FUNCTION_BLOCK FB_System_BSp_Ablaufsteuerung
VAR_IN_OUT
	Zustand					: ST_System_BSp_Zustand;
	Stellwert				: ST_System_BSp_Stellwert;
	Steuerung				: ST_System_BSp_Steuerung;
END_VAR
VAR_INPUT
	Zustand_Stellventil		: ST_SV_Zustand;
	Zustand_Pumpe			: ST_PU_Zustand;
	Zustand_Pumpe_Sp		: ST_PU_Schuetz_Zustand;
END_VAR
VAR_OUTPUT
END_VAR
VAR
END_VAR

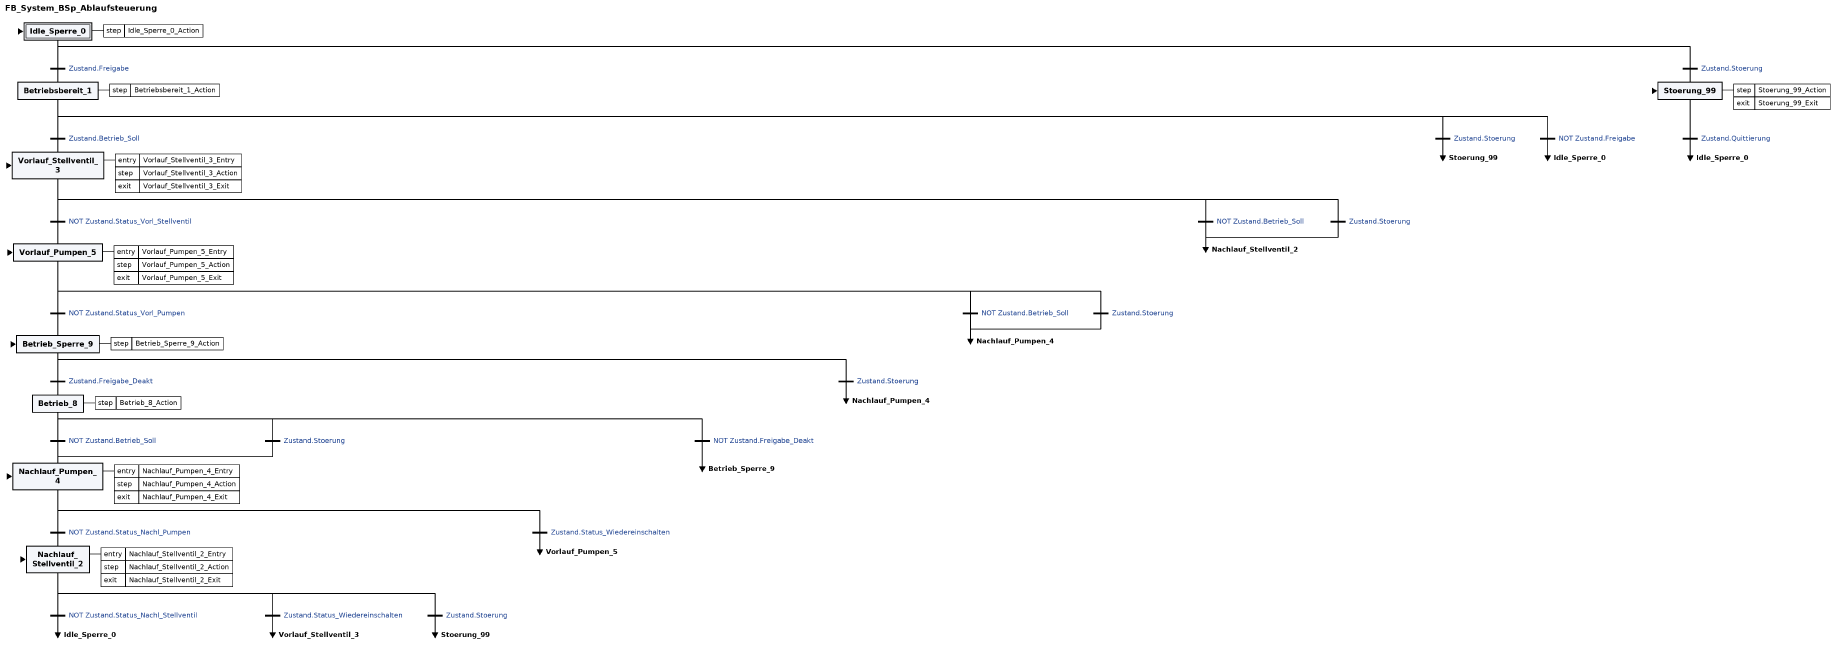
INITIAL_STEP Idle_Sperre_0:
    Idle_Sperre_0_Action(N);  // step action
END_STEP
TRANSITION FROM Idle_Sperre_0 TO Betriebsbereit_1
    := Zustand.Freigabe;
END_TRANSITION
TRANSITION FROM Idle_Sperre_0 TO Stoerung_99
    := Zustand.Stoerung;
END_TRANSITION
STEP Stoerung_99:
    Stoerung_99_Action(N);  // step action
    Stoerung_99_Exit(P0);  // exit action
END_STEP
TRANSITION FROM Stoerung_99 TO Idle_Sperre_0
    := Zustand.Quittierung;
END_TRANSITION
STEP Betriebsbereit_1:
    Betriebsbereit_1_Action(N);  // step action
END_STEP
TRANSITION FROM Betriebsbereit_1 TO Vorlauf_Stellventil_3
    := Zustand.Betrieb_Soll;
END_TRANSITION
TRANSITION FROM Betriebsbereit_1 TO Stoerung_99
    := Zustand.Stoerung;
END_TRANSITION
TRANSITION FROM Betriebsbereit_1 TO Idle_Sperre_0
    := NOT Zustand.Freigabe;
END_TRANSITION
STEP Vorlauf_Stellventil_3:
    Vorlauf_Stellventil_3_Entry(P1);  // entry action
    Vorlauf_Stellventil_3_Action(N);  // step action
    Vorlauf_Stellventil_3_Exit(P0);  // exit action
END_STEP
TRANSITION FROM Vorlauf_Stellventil_3 TO Vorlauf_Pumpen_5
    := NOT Zustand.Status_Vorl_Stellventil;
END_TRANSITION
TRANSITION FROM Vorlauf_Stellventil_3 TO Nachlauf_Stellventil_2
    := NOT Zustand.Betrieb_Soll;
END_TRANSITION
TRANSITION FROM Vorlauf_Stellventil_3 TO Nachlauf_Stellventil_2
    := Zustand.Stoerung;
END_TRANSITION
STEP Vorlauf_Pumpen_5:
    Vorlauf_Pumpen_5_Entry(P1);  // entry action
    Vorlauf_Pumpen_5_Action(N);  // step action
    Vorlauf_Pumpen_5_Exit(P0);  // exit action
END_STEP
TRANSITION FROM Vorlauf_Pumpen_5 TO Betrieb_Sperre_9
    := NOT Zustand.Status_Vorl_Pumpen;
END_TRANSITION
TRANSITION FROM Vorlauf_Pumpen_5 TO Nachlauf_Pumpen_4
    := NOT Zustand.Betrieb_Soll;
END_TRANSITION
TRANSITION FROM Vorlauf_Pumpen_5 TO Nachlauf_Pumpen_4
    := Zustand.Stoerung;
END_TRANSITION
STEP Betrieb_Sperre_9:
    Betrieb_Sperre_9_Action(N);  // step action
END_STEP
TRANSITION FROM Betrieb_Sperre_9 TO Betrieb_8
    := Zustand.Freigabe_Deakt;
END_TRANSITION
TRANSITION FROM Betrieb_Sperre_9 TO Nachlauf_Pumpen_4
    := Zustand.Stoerung;
END_TRANSITION
STEP Betrieb_8:
    Betrieb_8_Action(N);  // step action
END_STEP
TRANSITION FROM Betrieb_8 TO Nachlauf_Pumpen_4
    := NOT Zustand.Betrieb_Soll;
END_TRANSITION
TRANSITION FROM Betrieb_8 TO Nachlauf_Pumpen_4
    := Zustand.Stoerung;
END_TRANSITION
TRANSITION FROM Betrieb_8 TO Betrieb_Sperre_9
    := NOT Zustand.Freigabe_Deakt;
END_TRANSITION
STEP Nachlauf_Pumpen_4:
    Nachlauf_Pumpen_4_Entry(P1);  // entry action
    Nachlauf_Pumpen_4_Action(N);  // step action
    Nachlauf_Pumpen_4_Exit(P0);  // exit action
END_STEP
TRANSITION FROM Nachlauf_Pumpen_4 TO Nachlauf_Stellventil_2
    := NOT Zustand.Status_Nachl_Pumpen;
END_TRANSITION
TRANSITION FROM Nachlauf_Pumpen_4 TO Vorlauf_Pumpen_5
    := Zustand.Status_Wiedereinschalten;
END_TRANSITION
STEP Nachlauf_Stellventil_2:
    Nachlauf_Stellventil_2_Entry(P1);  // entry action
    Nachlauf_Stellventil_2_Action(N);  // step action
    Nachlauf_Stellventil_2_Exit(P0);  // exit action
END_STEP
TRANSITION FROM Nachlauf_Stellventil_2 TO Idle_Sperre_0
    := NOT Zustand.Status_Nachl_Stellventil;
END_TRANSITION
TRANSITION FROM Nachlauf_Stellventil_2 TO Vorlauf_Stellventil_3
    := Zustand.Status_Wiedereinschalten;
END_TRANSITION
TRANSITION FROM Nachlauf_Stellventil_2 TO Stoerung_99
    := Zustand.Stoerung;
END_TRANSITION

ACTION Betrieb_8_Action:
(* Stellwert setzen *)
Stellwert.Anford_Stellventil	:= TRUE;
Stellwert.Anford_Pumpe			:= TRUE;
Stellwert.Anford_Pumpe_Sp		:= TRUE;

(* Zustand setzen *)
Zustand.Status					:= E_System_BSp_Zustand_Status_Betrieb;
END_ACTION

ACTION Betrieb_Sperre_9_Action:
(* Stellwert setzen *)
Stellwert.Anford_Stellventil		:= TRUE;
Stellwert.Anford_Pumpe		:= TRUE;
Stellwert.Anford_Pumpe_Sp		:= TRUE;

(* Zustand setzen *)
Zustand.Status				:= E_System_BSp_Zustand_Status_Betrieb_Sperre;
END_ACTION

ACTION Betriebsbereit_1_Action:
(* Stellwert setzen *)
Stellwert.Anford_Stellventil	:= FALSE;
Stellwert.Anford_Pumpe			:= FALSE;
Stellwert.Anford_Pumpe_Sp		:= FALSE;

(* Zustand setzen *)
Zustand.Status			:= E_System_BSp_Zustand_Status_Betriebsbereit;
END_ACTION

ACTION Idle_Sperre_0_Action:
(* Stellwert setzen *)
Stellwert.Anford_Stellventil		:= FALSE;
Stellwert.Anford_Pumpe		:= FALSE;
Stellwert.Anford_Pumpe_Sp		:= FALSE;

(* Zustand setzen *)
Zustand.Status				:= E_System_BSp_Zustand_Status_Idle_Sperre;

(* Quittierungszustand auf False setzen, damit das System bei einer erneuten Störung nicht direkt wieder angeschaltet wird *)
Steuerung.Quittierung	:= FALSE;
END_ACTION

ACTION Nachlauf_Pumpen_4_Action:
(* Stellwert setzen *)
Stellwert.Anford_Stellventil	:= FALSE;
Stellwert.Anford_Pumpe			:= FALSE;
Stellwert.Anford_Pumpe_Sp		:= FALSE;

(* Zustand setzen *)
Zustand.Status				:= E_System_BSp_Zustand_Status_Nachl_Pumpen;
Zustand.Status_Nachl_Pumpen	:= Zustand_Pumpe.Betrieb OR Zustand_Pumpe_Sp.Betrieb OR Zustand_Pumpe.Status_Nachl OR Zustand_Pumpe_Sp.Status_Nachl;
Zustand.Status_Wiedereinschalten := Zustand.Betrieb_Soll AND Stellwert.Einschalten;
END_ACTION

ACTION Nachlauf_Pumpen_4_Entry:
Zustand.Status_Nachl_Pumpen	:= TRUE;
END_ACTION

ACTION Nachlauf_Pumpen_4_Exit:
Zustand.Status_Nachl_Pumpen	:= FALSE;
END_ACTION

ACTION Nachlauf_Stellventil_2_Action:
(* Stellwert setzen *)
Stellwert.Anford_Stellventil		:= FALSE;
Stellwert.Anford_Pumpe		:= FALSE;
Stellwert.Anford_Pumpe_Sp		:= FALSE;

(* Zustand setzen *)
Zustand.Status				:= E_System_BSp_Zustand_Status_Nachl_Stellventil;
Zustand.Status_Nachl_Stellventil	:= Zustand_Stellventil.Stellung OR Zustand_Stellventil.Stellungwechsel10;
Zustand.Status_Wiedereinschalten := Zustand.Betrieb_Soll AND Stellwert.Einschalten;
END_ACTION

ACTION Nachlauf_Stellventil_2_Entry:
Zustand.Status_Nachl_Stellventil	:= TRUE;
END_ACTION

ACTION Nachlauf_Stellventil_2_Exit:
Zustand.Status_Nachl_Stellventil	:= FALSE;
END_ACTION

ACTION Stoerung_99_Action:
(* Stellwert setzen *)
Stellwert.Anford_Stellventil	:= FALSE;
Stellwert.Anford_Pumpe			:= FALSE;
Stellwert.Anford_Pumpe_Sp		:= FALSE;

(* Zustand setzen *)
Zustand.Stoerung				:= TRUE;
Zustand.Status					:= E_System_BSp_Zustand_Status_Stoerung;
END_ACTION

ACTION Stoerung_99_Exit:
Zustand.Stoerung	:= FALSE;
END_ACTION

ACTION Vorlauf_Pumpen_5_Action:
(* Stellwert setzen *)
Stellwert.Anford_Stellventil		:= TRUE;
Stellwert.Anford_Pumpe		:= TRUE;
Stellwert.Anford_Pumpe_Sp		:= TRUE;

(* Zustand setzen *)
Zustand.Status				:= E_System_BSp_Zustand_Status_Vorl_Pumpen;
Zustand.Status_Vorl_Pumpen	:= NOT(Zustand_Pumpe.Betrieb AND Zustand_Pumpe_Sp.Betrieb AND NOT Zustand_Pumpe.Status_Vorl AND NOT Zustand_Pumpe_Sp.Status_Vorl);
END_ACTION

ACTION Vorlauf_Pumpen_5_Entry:
Zustand.Status_Vorl_Pumpen	:= TRUE;
END_ACTION

ACTION Vorlauf_Pumpen_5_Exit:
Zustand.Status_Vorl_Pumpen	:= FALSE;
END_ACTION

ACTION Vorlauf_Stellventil_3_Action:
(* Stellwert setzen *)
Stellwert.Anford_Stellventil		:= TRUE;
Stellwert.Anford_Pumpe		:= FALSE;
Stellwert.Anford_Pumpe_Sp		:= FALSE;

(* Zustand setzen *)
Zustand.Status				:= E_System_BSp_Zustand_Status_Vorl_Stellventil;
Zustand.Status_Vorl_Stellventil	:= NOT(Zustand_Stellventil.Stellung AND NOT Zustand_Stellventil.Stellungwechsel01);
END_ACTION

ACTION Vorlauf_Stellventil_3_Entry:
Zustand.Status_Vorl_Stellventil	:= TRUE;
END_ACTION

ACTION Vorlauf_Stellventil_3_Exit:
Zustand.Status_Vorl_Stellventil	:= FALSE;
END_ACTION

END_FUNCTION_BLOCK

(* stored: Version 1.1.0.1, ProductVersion 3.1.4024.9
   POU FB_System_BSp_Ablaufsteuerung: Id {1b44faae-4f25-44cd-be4c-999ff2f5d263}, SpecialFunc None
   Action Betrieb_8_Action: Id {0ce3c809-5c21-4956-89ba-cf6a9e1fdca3}
   Action Betrieb_Sperre_9_Action: Id {c1114971-bdcc-4776-8539-c9d7c4a4bbb3}
   Action Betriebsbereit_1_Action: Id {0460251c-e1b6-4f4e-946e-8cef174eb685}
   Action Idle_Sperre_0_Action: Id {1ca70484-d28a-400d-8ed7-cacfaa5d8784}
   Action Nachlauf_Pumpen_4_Action: Id {59d6b337-d4c1-44d8-b45c-9cafd9831f30}
   Action Nachlauf_Pumpen_4_Entry: Id {2a3bc810-2cc8-4da9-aa22-062232cae627}
   Action Nachlauf_Pumpen_4_Exit: Id {5cbe94ae-1138-4388-ae56-3a6a1f9074ae}
   Action Nachlauf_Stellventil_2_Action: Id {e82f1d45-962c-4fe3-a246-757cb1e0ab84}
   Action Nachlauf_Stellventil_2_Entry: Id {a5e05e29-1531-4da8-ac25-43780d0e0766}
   Action Nachlauf_Stellventil_2_Exit: Id {a25d462a-ce01-4420-a043-057435257a2d}
   Action Stoerung_99_Action: Id {9400e8e1-9785-46fd-8206-0f3b4516eb14}
   Action Stoerung_99_Exit: Id {237a27ce-709d-4cc2-88b3-d403d72dced7}
   Action Vorlauf_Pumpen_5_Action: Id {d108f33a-76e6-400a-9c01-7b7a39880bff}
   Action Vorlauf_Pumpen_5_Entry: Id {2bd748de-b57b-4026-9a67-d3e77d659357}
   Action Vorlauf_Pumpen_5_Exit: Id {2b872e26-ace0-4031-84c4-9e7bf1d197a8}
   Action Vorlauf_Stellventil_3_Action: Id {e9ec929b-8821-4dfd-b1b2-008299638a46}
   Action Vorlauf_Stellventil_3_Entry: Id {b96973da-066d-4188-8ec2-a358967ff49d}
   Action Vorlauf_Stellventil_3_Exit: Id {dae1a574-a37c-4010-974f-fb86251a4ae6} *)
